(* PLC project Tc2_Utilities.TC_SysLatencyEx Demo, tc3-libraries-kb TwinCAT 3.1 *)
(* stored: creationDateTime 2026-05-11T00:00:00, modificationDateTime 2026-05-11T00:00:00 *)

PROGRAM P_Demo_TC_SysLatencyEx
  VAR
    fbTC_SysLatencyEx : TC_SysLatencyEx;  (* TC_SysLatencyEx 实例 *)
    bRead : BOOL := TRUE;
    nAct : UDINT;
    nMax : UDINT;
    nMin : UDINT;
    bBusy_ : BOOL;
    bErrFlag : BOOL;
    nErrCode : UDINT;
  END_VAR

// =============================================================================
// 场景：长期趋势分析。
// 价值：完整统计。
// 验证：触发后观察多个 latency 统计字段。
// 验证步骤：
//   1. 右键 PLC 项目 → Import PLCopenXML → 选本文件
//   2. 引用 Tc2_Utilities（References → Add library）
//   3. 编译 → 登录 → 运行；按上方『验证』行的指示在线写值观察
// =============================================================================

fbTC_SysLatencyEx(
    NETID := '', START := bRead, TMOUT := DEFAULT_ADS_TIMEOUT,
    BUSY => bBusy_, ERR => bErrFlag, ERRID => nErrCode
);
END_PROGRAM
